FUNCTION_BLOCK FB_HomeRoutine_CalibrationCam EXTENDS FB_CyclicFB IMPLEMENTS I_MotionSequence
VAR
	_Axis : I_BasicAxis;

	//
	MCHomeCalCam	: MC_Home;
	_HomingDn		: BOOL;
	SequenceStep	: UDINT;
	_Position		: LREAL;
	_Options		: ST_HomingOptions;
	_CalibrationCam : BOOL;
END_VAR

PROPERTY Axis : I_BasicAxis
GET
Axis := _Axis;
END_GET
SET
_Axis := Axis;
END_SET
END_PROPERTY

PROPERTY CalibrationCam : BOOL
GET
CalibrationCam := _CalibrationCam;
END_GET
SET
_CalibrationCam := CalibrationCam;
END_SET
END_PROPERTY

METHOD PUBLIC CyclicLogic
CASE SequenceStep OF
	10:
		MCHomeCalCam(Axis			 := _Axis.Axis,
					 Execute		 := TRUE,
					 Position		 := _Position,
					 HomingMode		 := MC_HomingMode.MC_DefaultHoming,
					 Options		 := _Options,
					 bCalibrationCam := _CalibrationCam);

		IF NOT MCHomeCalCam.Busy THEN
			IF MCHomeCalCam.Error THEN
				_Error		 := TRUE;
				_ErrorID	 := MCHomeCalCam.ErrorID;
				SequenceStep := 0;
			ELSE
				//No error occurred
				SequenceStep := 0;
			END_IF

			MCHomeCalCam(Axis := _Axis.Axis, Execute := FALSE);
		END_IF

	
END_CASE

_Busy := SequenceStep <> 0;
END_METHOD

METHOD Execute : BOOL
IF (_Axis = 0) OR _Busy THEN
	RETURN;
END_IF

_Busy		 := TRUE;
_Error		 := FALSE;
_ErrorID	 := 0;
_HomingDn	 := FALSE;
SequenceStep := 10;
Execute		 := TRUE;
END_METHOD

PROPERTY Options : ST_HomingOptions
GET
Options := _Options;
END_GET
SET
_Options := Options;
END_SET
END_PROPERTY

PROPERTY Position : lreal
GET
Position := _Position;
END_GET
SET
_Position := Position;
END_SET
END_PROPERTY

END_FUNCTION_BLOCK

(* stored: Version 1.1.0.1, ProductVersion 3.1.4024.13
   POU FB_HomeRoutine_CalibrationCam: Id {dbe5de1d-4390-49bb-bad5-fae195f2ce94}, SpecialFunc None
   Property Axis: Id {9307518c-53f9-08b1-15d4-18035b66ffa5}
   Get Get: Id {3178f8fd-1a56-08c5-3bd2-12ec58d8df5f}
   Set Set: Id {077dfdb4-eb73-0913-29f6-caea5df7f37d}
   Property CalibrationCam: Id {0ddd634d-37c3-4f62-90e4-9fa1ef7ddd66}
   Get Get: Id {512f6d08-e037-4cc7-977c-23ac5de197e3}
   Set Set: Id {43034147-9d46-4434-b718-2f73343803b7}
   Method CyclicLogic: Id {3b68e5be-7410-4a10-ba7e-73d4e8433cfc}
   Method Execute: Id {a6cb3749-21f6-4829-adcc-beccdb4982d3}
   Property Options: Id {ef04d79c-086d-4006-9a52-3584ed73a850}
   Get Get: Id {d1c0e72d-093f-4d90-980b-1de0392586d7}
   Set Set: Id {ad421931-833b-44fe-acf9-45ceb9fcdcc8}
   Property Position: Id {b90d3843-878d-483c-943e-a235c1193d64}
   Get Get: Id {e687b55a-6f98-4947-8a43-955859baacb9}
   Set Set: Id {afb6a16b-5efe-48a5-ac28-771b0afce150} *)
